# EPICS substitutions: EUROTHRM/EUROTHRM-IOC-01App/Db/devEurothrmA09.substitutions
# Note: this file is generated by generate_substitutions.py
file devEurothrm.template {
pattern { P, GAD, LAD, MODBUS_PV, MODBUS_SP, MODBUS_P, MODBUS_I, MODBUS_D, MODBUS_HS, MODBUS_LS, MODBUS_AT, MODBUS_HO, MODBUS_OP }
{ "\$(P)", "0", "9", "8193", "8194", "8198", "8200", "8201", "8303", "8304", "8462", "8222", "8195" }
}
